{attribute 'linkalways'} 
{attribute 'no_explicit_call' := 'This FB is a CLASS and must be accessed using methods or properties'}
{attribute 'enable_dynamic_creation'}
FUNCTION_BLOCK ServerResponse IMPLEMENTS I_ServerResponse
VAR
	_header : Header(0);
	_sent : BOOL := FALSE;
	responseData : ResponseData;
	headerAccessor : I_ServerResponseHeaderAccessor;
END_VAR

METHOD PUBLIC Accepted
VAR_INPUT
END_VAR
IF _sent THEN
	RETURN;
END_IF

headerAccessor.UpdateResponseWithAccepted(THIS^);
CompleteResponseWithoutPayload();
END_METHOD

METHOD PUBLIC Busy
VAR_INPUT
END_VAR
IF _sent THEN
	RETURN;
END_IF

headerAccessor.UpdateResponseWithBusy(THIS^);
CompleteResponseWithoutPayload();
END_METHOD

METHOD PRIVATE CompleteResponseWithoutPayload
VAR_INPUT
END_VAR
_sent := TRUE;
_header.ToString(responseData.Header);
memset(ADR(responseData.Payload),0,SIZEOF(responseData.Payload));
END_METHOD

METHOD PRIVATE CompleteResponseWithPayload
VAR_INPUT
	PayloadDataAddress : PVOID;
	PayloadDataSize : UDINT;
END_VAR
_sent := TRUE;
_header.ToString(responseData.Header);
memcpy(ADR(responseData.Payload),PayloadDataAddress,PayloadDataSize);
END_METHOD

METHOD PUBLIC Error
VAR_INPUT
	ErrorCode : T_MAXSTRING;
	Message : T_MAXSTRING;
END_VAR
IF _sent THEN
	RETURN;
END_IF

headerAccessor.UpdateResponseWithError(THIS^, ErrorCode, Message);
CompleteResponseWithoutPayload();
END_METHOD

METHOD FB_init : BOOL
VAR_INPUT
	bInitRetains : BOOL; // if TRUE, the retain variables are initialized (warm start / cold start)
	bInCopyCode : BOOL;  // if TRUE, the instance afterwards gets moved into the copy code (online change)
	HeaderAccessor : I_ServerResponseHeaderAccessor;
END_VAR
THIS^.headerAccessor := HeaderAccessor;
memset(ADR(responseData),0,SIZEOF(responseData));
END_METHOD

PROPERTY PUBLIC Header : I_Header
GET
Header := _header;
END_GET
END_PROPERTY

PROPERTY PUBLIC HeadersSent : BOOL
GET
HeadersSent := _sent;
END_GET
END_PROPERTY

METHOD PUBLIC Pending
VAR_INPUT
	ResponseId : REFERENCE TO T_MAXSTRING;
	RetryDelayInMs : UDINT;
END_VAR
IF _sent THEN
	RETURN;
END_IF

IF (NOT __ISVALIDREF(ResponseId)) OR_ELSE ResponseId = '' THEN
	Error('MISSING_RESPONSE_ID', 'Unable to mark response as pending without ResponseId');
	RETURN;
END_IF

headerAccessor.UpdateResponseWithPending(THIS^, ResponseId, RetryDelayInMs);
CompleteResponseWithoutPayload();
END_METHOD

METHOD PUBLIC Success
VAR_INPUT
END_VAR
VAR
	errorMessage : T_MAXSTRING;
END_VAR
IF _sent THEN
	RETURN;
END_IF

headerAccessor.UpdateResponseWithSuccess(THIS^);
CompleteResponseWithoutPayload();
END_METHOD

METHOD PUBLIC SuccessWithPayload
VAR_INPUT
	PayloadDataAddress : PVOID;
	PayloadDataSize : UDINT;
END_VAR
VAR
	errorMessage : T_MAXSTRING;
	maximumPayloadDataSize : UDINT;
END_VAR
IF _sent THEN
	RETURN;
END_IF

// SIZEOF includes the null terminator, which must stay within the buffer,
// so only SIZEOF - 1 bytes of actual payload data can be transmitted.
maximumPayloadDataSize := SIZEOF(responseData.Payload) - 1;

IF PayloadDataSize > maximumPayloadDataSize THEN
	errorMessage := 'Payload too big to transmit. Maximum : ';
	errorMessage := concat(errorMessage, UDINT_TO_STRING(maximumPayloadDataSize));
	errorMessage := concat(errorMessage, ', Actual Size : ');
	errorMessage := concat(errorMessage, UDINT_TO_STRING(PayloadDataSize));
	Error('PAYLOAD_TOO_BIG', errorMessage);
	RETURN;
END_IF

headerAccessor.UpdateResponseWithSuccess(THIS^);
CompleteResponseWithPayload(PayloadDataAddress, PayloadDataSize);
END_METHOD

METHOD PUBLIC TryGetData : BOOL;
VAR_INPUT
	Destination : REFERENCE TO ResponseData;
END_VAR
IF NOT __ISVALIDREF(Destination) THEN
	RETURN;
END_IF

IF SIZEOF(Destination) <> SIZEOF(responseData) THEN
	RETURN;
END_IF

memcpy(ADR(Destination), ADR(responseData), SIZEOF(Destination));
TryGetData := TRUE;
END_METHOD

END_FUNCTION_BLOCK

(* stored: Version 1.1.0.1, ProductVersion 3.1.4026.18
   POU ServerResponse: Id {2442627d-7496-4f6b-af53-517e3869f380}, SpecialFunc None
   Folder Constructor: Id {e8cbe832-724d-4258-9644-602186047960}
   Folder Private: Id {02b7177e-0c8a-4f2a-a25b-c679e3130a56}
   Method Accepted: Id {6e56c744-dca2-49fb-81f6-ab1642a8984b}
   Method Busy: Id {1e41d8c7-d402-4fda-a0ff-e7e6a9830755}
   Method CompleteResponseWithoutPayload: Id {c9a20195-b63c-4cf1-9d9b-954c8e05178f}
   Method CompleteResponseWithPayload: Id {0d2d7ff9-4809-431c-984c-e6ae3599afb3}
   Method Error: Id {999d566d-2849-4be7-a7f2-4a38bbc0bfe3}
   Method FB_init: Id {75613d85-36a0-483f-9cb9-b153a4a35fec}
   Property Header: Id {0fa71884-bf67-4292-8a3e-e8f67c31637d}
   Get Get: Id {a88d816b-b864-488b-8dc3-acf657eb04c1}
   Property HeadersSent: Id {29bf1bda-2f1e-43a3-b208-2c3514b2b8a0}
   Get Get: Id {9d97eeba-a138-41f0-bad4-6b5e2d32884b}
   Method Pending: Id {2874985b-49d4-4b31-9a4e-3f0794be3590}
   Method Success: Id {94c7cca4-6ca8-4833-80e2-753569bcce1e}
   Method SuccessWithPayload: Id {0b1ed937-31ec-4ff5-b481-0ec496f95421}
   Method TryGetData: Id {b5dfab8d-70d8-4594-8c15-b16db1a82e29} *)
